INTERFACE ITF_XTSIOEnvVarWrapper

METHOD GetCaGroupInterface : I_Mc2CaGroup
VAR_INPUT
	CAGroupNumber : INT;
END_VAR
END_METHOD

METHOD PUBLIC GetMotorModuleInterface : I_TcIoXtsPartModule
VAR_INPUT
	PartNumber : INT;
	ModuleNumber : INT;
END_VAR
END_METHOD

METHOD PUBLIC GetMoverInterface : I_TcIoXtsXpuMover
VAR_INPUT
	MoverId : INT;
END_VAR
END_METHOD

METHOD PUBLIC GetPartInterface : I_TcIoXtsXpuPart
VAR_INPUT
	PartNumber : INT;
END_VAR
END_METHOD

METHOD PUBLIC GetTrackInterface : I_TcIoXtsXpuTrack
VAR_INPUT
	TrackNumber : INT;
END_VAR
END_METHOD

END_INTERFACE

(* stored: Version 1.1.0.1, ProductVersion 3.1.4024.12
   Itf ITF_XTSIOEnvVarWrapper: Id {30a06d50-ef59-4bfa-9dd3-f949d401bfcc}
   Method GetCaGroupInterface: Id {e5766ff7-d74d-4918-8c8c-b6404824695c}
   Method GetMotorModuleInterface: Id {c9e316a7-456a-49d5-b1f4-827c270545da}
   Method GetMoverInterface: Id {30f73f3d-ac87-4263-a943-1883fb33de68}
   Method GetPartInterface: Id {33ed9cb1-a852-4796-a6f8-db3ef7d84470}
   Method GetTrackInterface: Id {46ac4c9d-e2d5-4696-a8bf-e6e5f3db6a25} *)
